// Mitsubishi GX Works2 project: BookEX6_29 Other   PLC: Q13UDV

// global labels: Global
VAR_GLOBAL
  bVar0 AT M5000 : BOOL;
  abArray0 AT M5010 : ARRAY [0..49] OF BOOL;
  sStr0 AT D5000 : STRING[199];
  sStr1 AT D5100 : STRING[199];
  sStr2 AT D5200 : STRING[199];
  sStr3 AT D5300 : STRING[199];
  sStr4 AT D5400 : STRING[199];
  sStr5 AT D5500 : STRING[199];
  sStr6 AT D5600 : STRING[199];
  sStr7 AT D5700 : STRING[199];
  sStr8 AT D5800 : STRING[199];
  sStr9 AT D5900 : STRING[199];
  iVar0 AT D4500 : INT;
  iVar1 AT D4501 : INT;
  iVar2 AT D4502 : INT;
  iVar3 AT D4503 : INT;
  iVar4 AT D4504 : INT;
  iVar5 AT D4505 : INT;
  iVar6 AT D4506 : INT;
  iVar7 AT D4507 : INT;
  iVar8 AT D4508 : INT;
  iVar9 AT D4509 : INT;
  dVar0 AT D4510 : DINT;
  dVar1 AT D4512 : DINT;
  dVar2 AT D4514 : DINT;
  dVar3 AT D4516 : DINT;
  dVar4 AT D4518 : DINT;
  dVar5 AT D4520 : DINT;
  dVar6 AT D4522 : DINT;
  dVar7 AT D4524 : DINT;
  dVar8 AT D4526 : DINT;
  dVar9 AT D4528 : DINT;
  wVar0 AT D4530 : WORD;
  wVar1 AT D4531 : WORD;
  wVar2 AT D4532 : WORD;
  wVar3 AT D4533 : WORD;
  wVar4 AT D4534 : WORD;
  wVar5 AT D4535 : WORD;
  wVar6 AT D4536 : WORD;
  wVar7 AT D4537 : WORD;
  wVar8 AT D4538 : WORD;
  wVar9 AT D4539 : WORD;
  dwVar0 AT D4540 : DWORD;
  dwVar1 AT D4542 : DWORD;
  dwVar2 AT D4544 : DWORD;
  dwVar3 AT D4546 : DWORD;
  dwVar4 AT D4548 : DWORD;
  dwVar5 AT D4550 : DWORD;
  dwVar6 AT D4552 : DWORD;
  dwVar7 AT D4554 : DWORD;
  dwVar8 AT D4556 : DWORD;
  dwVar9 AT D4558 : DWORD;
  fsVar0 AT D4560 : REAL;
  fsVar1 AT D4562 : REAL;
  fsVar2 AT D4564 : REAL;
  fsVar3 AT D4566 : REAL;
  fsVar4 AT D4568 : REAL;
  fsVar5 AT D4570 : REAL;
  fsVar6 AT D4572 : REAL;
  fsVar7 AT D4574 : REAL;
  fsVar8 AT D4576 : REAL;
  fsVar9 AT D4578 : REAL;
  fdVar0 AT D4580 : LREAL;
  tTime0 AT D4620 : TIME;
  tTime1 AT D4622 : TIME;
  tTime2 AT D4624 : TIME;
  tTime3 AT D4626 : TIME;
  tTime4 AT D4628 : TIME;
  tTime5 AT D4630 : TIME;
  tTime6 AT D4632 : TIME;
  tTime7 AT D4634 : TIME;
  tTime8 AT D4636 : TIME;
  tTime9 AT D4638 : TIME;
  tTime10 AT D4640 : TIME;
  bVar1 AT M5001 : BOOL;
  bVar2 AT M5002 : BOOL;
  bVar3 AT M5003 : BOOL;
  bVar4 AT M5004 : BOOL;
  bVar5 AT M5005 : BOOL;
  bVar6 AT M5006 : BOOL;
  bVar7 AT M5007 : BOOL;
  bVar8 AT M5008 : BOOL;
  bVar9 AT M5009 : BOOL;
  abArray1 AT M5060 : ARRAY [0..49] OF BOOL;
  abArray2 AT M5110 : ARRAY [0..49] OF BOOL;
  abArray3 AT M5160 : ARRAY [0..49] OF BOOL;
  abArray4 AT M5210 : ARRAY [0..49] OF BOOL;
  abArray5 AT M5260 : ARRAY [0..49] OF BOOL;
  abArray6 AT M5310 : ARRAY [0..49] OF BOOL;
  abArray7 AT M5360 : ARRAY [0..49] OF BOOL;
  abArray8 AT M5410 : ARRAY [0..49] OF BOOL;
  abArray9 AT M5460 : ARRAY [0..49] OF BOOL;
  fdVar1 AT D4584 : LREAL;
  fdVar2 AT D4588 : LREAL;
  fdVar3 AT D4592 : LREAL;
  fdVar4 AT D4596 : LREAL;
  fdVar5 AT D4600 : LREAL;
  fdVar6 AT D4604 : LREAL;
  fdVar7 AT D4608 : LREAL;
  fdVar8 AT D4612 : LREAL;
  fdVar9 AT D4616 : LREAL;
  afsPen0 AT D2000 : ARRAY [0..499] OF REAL;
  afsPen1 AT D3000 : ARRAY [0..499] OF REAL;
  abInp1 AT X10 : ARRAY [0..1] OF BOOL;
  abInp2 AT X12 : ARRAY [0..1] OF BOOL;
  adwD10 AT D10 : ARRAY [0..9] OF DWORD;
  awD10 AT D10 : ARRAY [0..19] OF WORD;
  abM10 AT M10 : ARRAY [0..19] OF BOOL;
END_VAR
// user libraries (not included): HMI

FUNCTION newENCO
VAR_INPUT
  w_IN : WORD;
END_VAR
VAR
  ix : INT;
  wTmp : WORD;
  iy : INT;
END_VAR
;
wTmp := H0001;
iy := 1;
FOR ix := 0 TO 15 DO 
	IF (w_IN AND wTmp) <> 0 THEN
		EXIT;
	END_IF;
	ROL(TRUE, 1, wTmp);
	iy := iy + 1;
END_FOR;
IF ix = 16 THEN
	iy := 0;
END_IF;
newENCO := iy;
END_FUNCTION

FUNCTION_BLOCK UpDw
VAR_INPUT
  b_CH1 : BOOL;
  b_CH2 : BOOL;
  b_RST : BOOL;
END_VAR
VAR_OUTPUT
  b_DIR : BOOL;
  i_Cnt : INT;
END_VAR
VAR
  bOld1 : BOOL;
  bOld2 : BOOL;
  bClk : BOOL;
  bClk1 : BOOL;
  baxb : BOOL;
  bClk2 : BOOL;
END_VAR
;
baxb := b_CH1 XOR b_CH2;
bClk1 := b_CH1 XOR bOld1;
bOld1 := b_CH1;
bClk2 := b_CH2 XOR bOld2;
bOld2 := b_CH2;
bClk := bClk1 OR bClk2;

IF baxb AND bClk1 THEN b_DIR := TRUE; END_IF;
IF baxb AND bClk2 THEN b_DIR := FALSE; END_IF;

IF bClk AND b_DIR THEN i_Cnt := i_Cnt + 1; END_IF;
IF bClk AND NOT b_DIR THEN i_Cnt := i_Cnt -1; END_IF;

IF b_RST THEN i_Cnt := 0; END_IF;
END_FUNCTION_BLOCK

PROGRAM Ex
(* structured ladder/FBD written out as ST: instructions are called as NAME(EN, inputs, outputs); _pN, _eN, _tN stand for wires *)
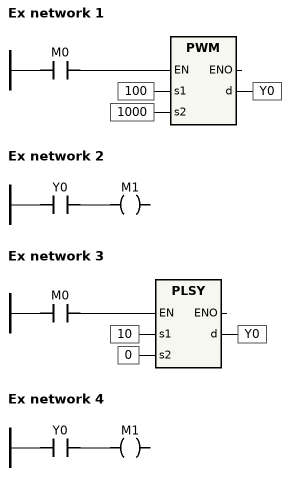
(* network 1 *)
PWM(M0, 100, 1000, Y0);
(* network 2 *)
M1 := Y0;
(* network 3 *)
PLSY(M0, 10, 0, Y0);
(* network 4 *)
M1 := Y0;
END_PROGRAM

PROGRAM ExMTR
(* structured ladder/FBD written out as ST: instructions are called as NAME(EN, inputs, outputs); _pN, _eN, _tN stand for wires *)
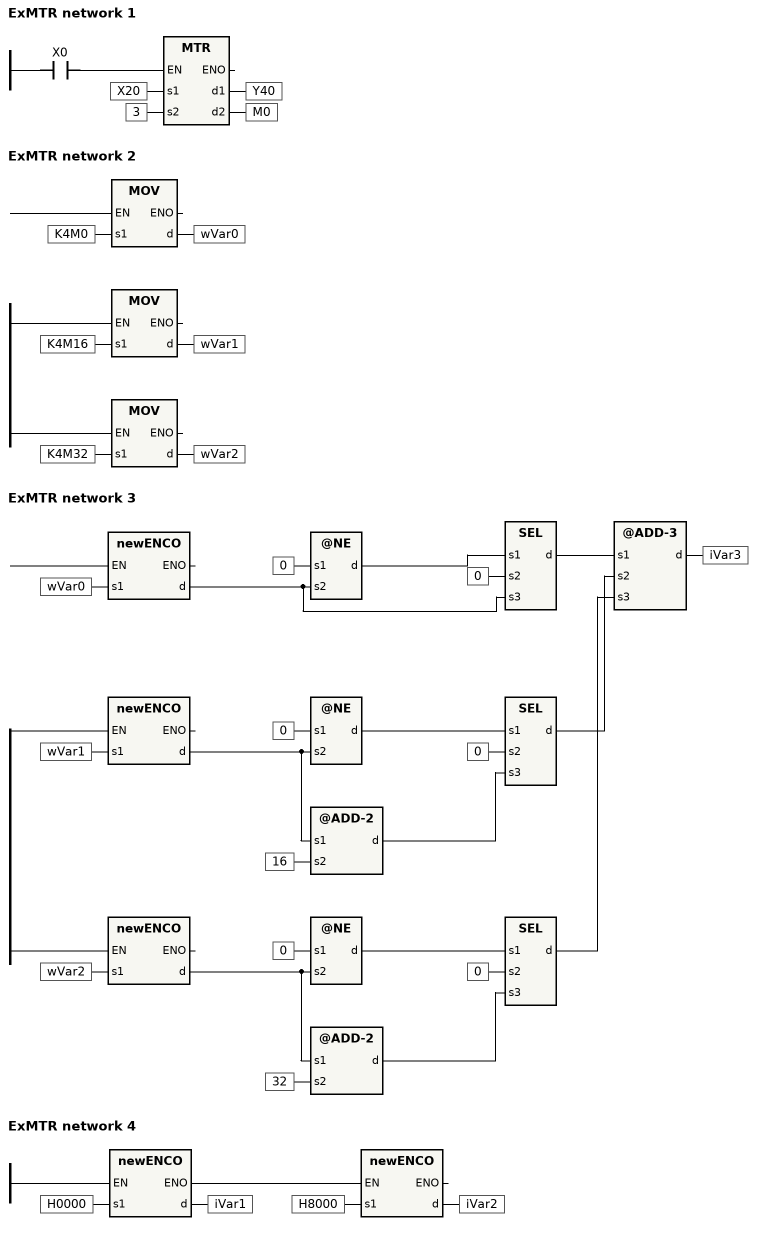
(* network 1 *)
MTR(X0, X20, 3, Y40, M0);
(* network 2 *)
MOV(TRUE, K4M0, wVar0);
MOV(TRUE, K4M16, wVar1);
MOV(TRUE, K4M32, wVar2);
(* network 3 *)
newENCO(TRUE, wVar0, _t1);
newENCO(TRUE, wVar1, _t2);
newENCO(TRUE, wVar2, _t3);
iVar3 := @ADD-3(SEL(@NE(0, _t1), 0, _t1), SEL(@NE(0, _t2), 0, @ADD-2(_t2, 16)), SEL(@NE(0, _t3), 0, @ADD-2(_t3, 32)));
(* network 4 *)
_e1 := newENCO(TRUE, H0000, iVar1);
newENCO(_e1, H8000, iVar2);
END_PROGRAM

PROGRAM ExPLSY
VAR
  HMI05_1 : HMI05;
END_VAR
(* structured ladder/FBD written out as ST: instructions are called as NAME(EN, inputs, outputs); _pN, _eN, _tN stand for wires *)
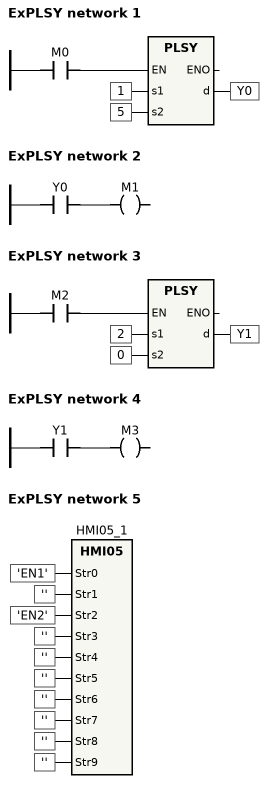
(* network 1 *)
PLSY(M0, 1, 5, Y0);
(* network 2 *)
M1 := Y0;
(* network 3 *)
PLSY(M2, 2, 0, Y1);
(* network 4 *)
M3 := Y1;
(* network 5 *)
HMI05_1(Str0 := 'EN1', Str1 := '', Str2 := 'EN2', Str3 := '', Str4 := '', Str5 := '', Str6 := '', Str7 := '', Str8 := '', Str9 := '');
END_PROGRAM

PROGRAM ExPWM
VAR
  HMI05_1 : HMI05;
  bFeed : BOOL;
  TON_HIGH_E_1 : TON_HIGH_E;
  TON_HIGH_E_2 : TON_HIGH_E;
END_VAR
(* structured ladder/FBD written out as ST: instructions are called as NAME(EN, inputs, outputs); _pN, _eN, _tN stand for wires *)
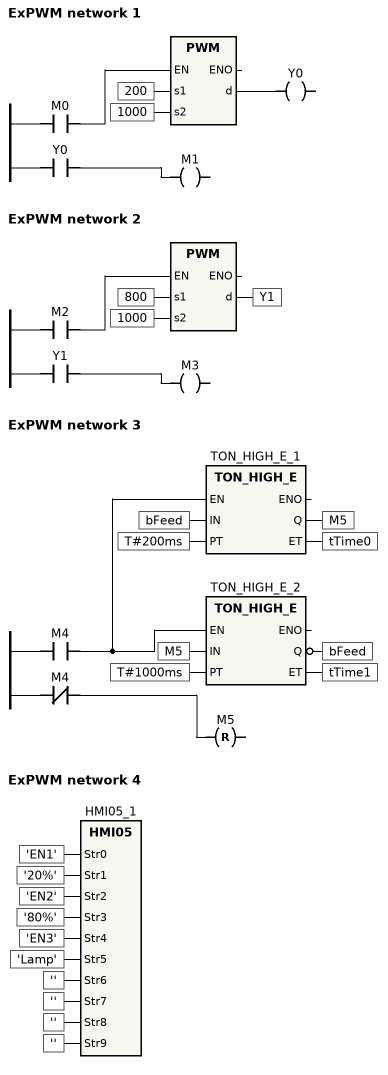
(* network 1 *)
PWM(M0, 200, 1000, _t1);
Y0 := _t1;
M1 := Y0;
(* network 2 *)
PWM(M2, 800, 1000, Y1);
M3 := Y1;
(* network 3 *)
TON_HIGH_E_1(EN := M4, IN := bFeed, PT := T#200ms, Q => M5, ET => tTime0);
TON_HIGH_E_2(EN := M4, IN := M5, PT := T#1000ms, ET => tTime1);
bFeed := NOT TON_HIGH_E_2.Q;
RST(NOT M4, M5);
(* network 4 *)
HMI05_1(Str0 := 'EN1', Str1 := '20%', Str2 := 'EN2', Str3 := '80%', Str4 := 'EN3', Str5 := 'Lamp', Str6 := '', Str7 := '', Str8 := '', Str9 := '');
END_PROGRAM

PROGRAM ExRAMP
VAR
  aiVar0 : ARRAY [0..1] OF INT;
  abRes3 : ARRAY [0..1] OF BOOL;
  HMI03_1 : HMI03;
END_VAR
(* structured ladder/FBD written out as ST: instructions are called as NAME(EN, inputs, outputs); _pN, _eN, _tN stand for wires *)
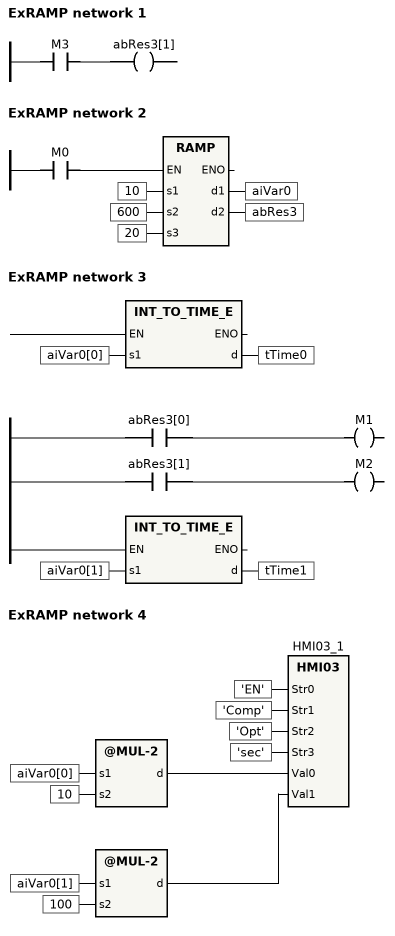
(* network 1 *)
abRes3[1] := M3;
(* network 2 *)
RAMP(M0, 10, 600, 20, aiVar0, abRes3);
(* network 3 *)
INT_TO_TIME_E(TRUE, aiVar0[0], tTime0);
INT_TO_TIME_E(TRUE, aiVar0[1], tTime1);
M1 := abRes3[0];
M2 := abRes3[1];
(* network 4 *)
HMI03_1(Str0 := 'EN', Str1 := 'Comp', Str2 := 'Opt', Str3 := 'sec', Val0 := @MUL-2(aiVar0[0], 10), Val1 := @MUL-2(aiVar0[1], 100));
END_PROGRAM

PROGRAM ExROTC
VAR
  aiVar2 : ARRAY [0..2] OF INT;
  abRes2 : ARRAY [0..7] OF BOOL;
  HMI05_1 : HMI05;
END_VAR
(* structured ladder/FBD written out as ST: instructions are called as NAME(EN, inputs, outputs); _pN, _eN, _tN stand for wires *)
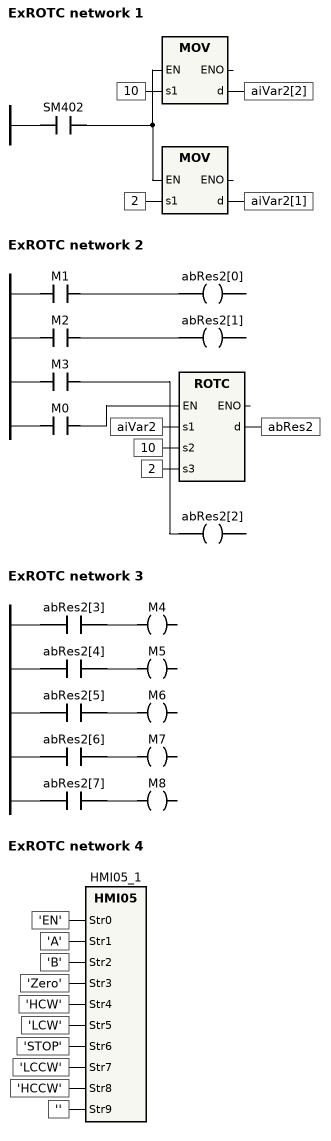
(* network 1 *)
MOV(SM402, 10, aiVar2[2]);
MOV(SM402, 2, aiVar2[1]);
(* network 2 *)
abRes2[0] := M1;
abRes2[1] := M2;
abRes2[2] := M3;
ROTC(M0, aiVar2, 10, 2, abRes2);
(* network 3 *)
M4 := abRes2[3];
M5 := abRes2[4];
M6 := abRes2[5];
M7 := abRes2[6];
M8 := abRes2[7];
(* network 4 *)
HMI05_1(Str0 := 'EN', Str1 := 'A', Str2 := 'B', Str3 := 'Zero', Str4 := 'HCW', Str5 := 'LCW', Str6 := 'STOP', Str7 := 'LCCW', Str8 := 'HCCW', Str9 := '');
END_PROGRAM

PROGRAM ExSPD
VAR
  HMI03_1 : HMI03;
END_VAR
(* structured ladder/FBD written out as ST: instructions are called as NAME(EN, inputs, outputs); _pN, _eN, _tN stand for wires *)
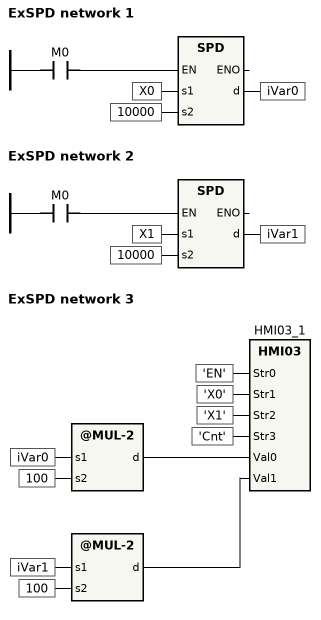
(* network 1 *)
SPD(M0, X0, 10000, iVar0);
(* network 2 *)
SPD(M0, X1, 10000, iVar1);
(* network 3 *)
HMI03_1(Str0 := 'EN', Str1 := 'X0', Str2 := 'X1', Str3 := 'Cnt', Val0 := @MUL-2(iVar0, 100), Val1 := @MUL-2(iVar1, 100));
END_PROGRAM

PROGRAM ExSTMR
VAR
  HMI05_1 : HMI05;
  abRes1 : ARRAY [0..3] OF BOOL;
END_VAR
(* structured ladder/FBD written out as ST: instructions are called as NAME(EN, inputs, outputs); _pN, _eN, _tN stand for wires *)
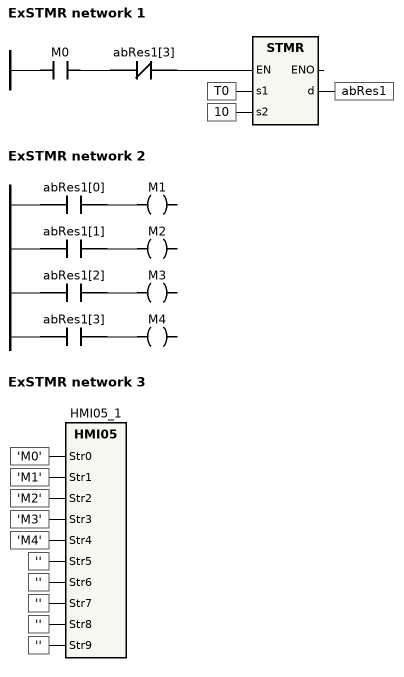
(* network 1 *)
STMR(M0 AND NOT abRes1[3], T0, 10, abRes1);
(* network 2 *)
M1 := abRes1[0];
M2 := abRes1[1];
M3 := abRes1[2];
M4 := abRes1[3];
(* network 3 *)
HMI05_1(Str0 := 'M0', Str1 := 'M1', Str2 := 'M2', Str3 := 'M3', Str4 := 'M4', Str5 := '', Str6 := '', Str7 := '', Str8 := '', Str9 := '');
END_PROGRAM

PROGRAM ExTTMR2
VAR
  aiVar0 : ARRAY [0..1] OF INT;
  HMI03_1 : HMI03;
  TTMR2_1 : TTMR2;
END_VAR
(* structured ladder/FBD written out as ST: instructions are called as NAME(EN, inputs, outputs); _pN, _eN, _tN stand for wires *)
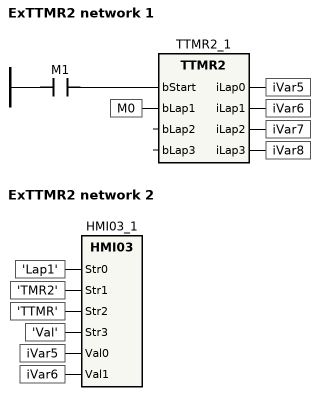
(* network 1 *)
TTMR2_1(bStart := M1, bLap1 := M0, iLap0 => iVar5, iLap1 => iVar6, iLap2 => iVar7, iLap3 => iVar8);
(* network 2 *)
HMI03_1(Str0 := 'Lap1', Str1 := 'TMR2', Str2 := 'TTMR', Str3 := 'Val', Val0 := iVar5, Val1 := iVar6);
END_PROGRAM

PROGRAM ExUDCNT
VAR
  HMI04_1 : HMI04;
END_VAR
(* structured ladder/FBD written out as ST: instructions are called as NAME(EN, inputs, outputs); _pN, _eN, _tN stand for wires *)
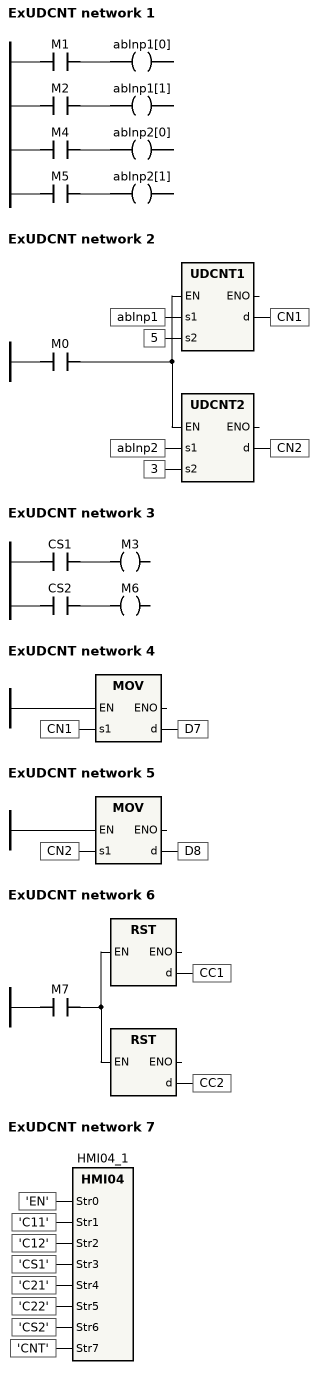
(* network 1 *)
abInp1[0] := M1;
abInp1[1] := M2;
abInp2[0] := M4;
abInp2[1] := M5;
(* network 2 *)
UDCNT1(M0, abInp1, 5, CN1);
UDCNT2(M0, abInp2, 3, CN2);
(* network 3 *)
M3 := CS1;
M6 := CS2;
(* network 4 *)
MOV(TRUE, CN1, D7);
(* network 5 *)
MOV(TRUE, CN2, D8);
(* network 6 *)
RST(M7, CC1);
RST(M7, CC2);
(* network 7 *)
HMI04_1(Str0 := 'EN', Str1 := 'C11', Str2 := 'C12', Str3 := 'CS1', Str4 := 'C21', Str5 := 'C22', Str6 := 'CS2', Str7 := 'CNT');
END_PROGRAM

PROGRAM ExUpDw
VAR
  HMI04_1 : HMI04;
  UpDw_1 : UpDw;
END_VAR
(* structured ladder/FBD written out as ST: instructions are called as NAME(EN, inputs, outputs); _pN, _eN, _tN stand for wires *)
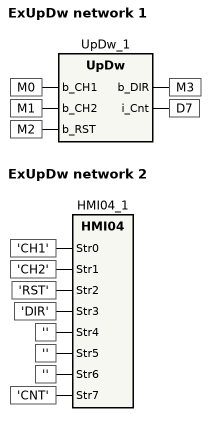
(* network 1 *)
UpDw_1(b_CH1 := M0, b_CH2 := M1, b_RST := M2, b_DIR => M3, i_Cnt => D7);
(* network 2 *)
HMI04_1(Str0 := 'CH1', Str1 := 'CH2', Str2 := 'RST', Str3 := 'DIR', Str4 := '', Str5 := '', Str6 := '', Str7 := 'CNT');
END_PROGRAM

PROGRAM ExTTMR
VAR
  aiVar0 : ARRAY [0..1] OF INT;
  HMI03_1 : HMI03;
  aiVar1 : ARRAY [0..1] OF INT;
END_VAR
(* structured ladder/FBD written out as ST: instructions are called as NAME(EN, inputs, outputs); _pN, _eN, _tN stand for wires *)
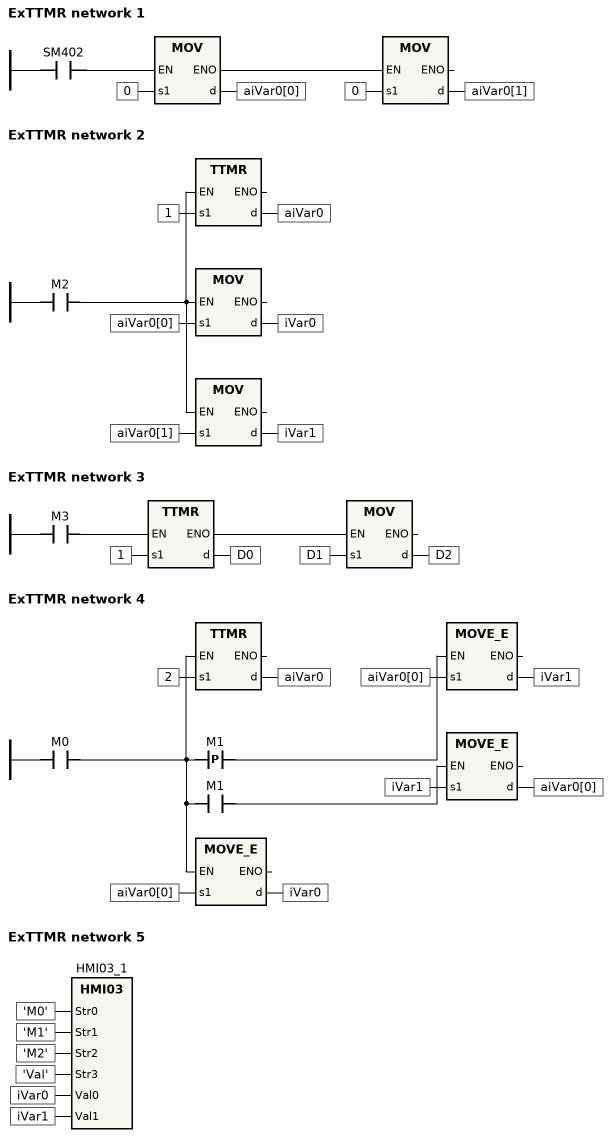
(* network 1 *)
_e1 := MOV(SM402, 0, aiVar0[0]);
MOV(_e1, 0, aiVar0[1]);
(* network 2 *)
TTMR(M2, 1, aiVar0);
MOV(M2, aiVar0[0], iVar0);
MOV(M2, aiVar0[1], iVar1);
(* network 3 *)
_e1 := TTMR(M3, 1, D0);
MOV(_e1, D1, D2);
(* network 4 *)
TTMR(M0, 2, aiVar0);
MOVE_E(M0, aiVar0[0], iVar0);
MOVE_E(M0 AND LDP(TRUE, M1), aiVar0[0], iVar1);
MOVE_E(M0 AND M1, iVar1, aiVar0[0]);
(* network 5 *)
HMI03_1(Str0 := 'M0', Str1 := 'M1', Str2 := 'M2', Str3 := 'Val', Val0 := iVar0, Val1 := iVar1);
END_PROGRAM

FUNCTION_BLOCK TTMR2
VAR_INPUT
  bStart : BOOL;
  bLap1 : BOOL;
  bLap2 : BOOL;
END_VAR
VAR_OUTPUT
  iLap0 : INT;
  iLap1 : INT;
  iLap2 : INT;
END_VAR
VAR
  dTime0 : DINT;
  dTime1 : DINT;
  dTime2 : DINT;
  dTmp : DINT;
END_VAR
VAR_OUTPUT
  iLap3 : INT;
END_VAR
VAR_INPUT
  bLap3 : BOOL;
END_VAR
VAR
  dTime3 : DINT;
END_VAR
;
IF LDP(TRUE, bStart) THEN
	dTime0 := 0;
	dTime1 := 0;
	dTime2 := 0;
	dTime3 := 0;
END_IF;
IF bStart THEN
	dTmp := INT_TO_DINT(SD520) *1000 + INT_TO_DINT(SD521);	
	dTime0 := dTime0 + dTmp;	
	IF LDP(TRUE, bLap1) THEN
		dTime1 := dTime0;
	END_IF;
	IF LDP(TRUE, bLap2) THEN
		dTime2 := dTime0;
	END_IF;
	IF LDP(TRUE, bLap3) THEN
		dTime3 := dTime0;
	END_IF;
END_IF;
iLap0 := DINT_TO_INT(dTime0 / 10000);	
iLap1 := DINT_TO_INT(dTime1 / 10000);
iLap2 := DINT_TO_INT(dTime2 / 10000);
iLap3 := DINT_TO_INT(dTime3 / 10000);
END_FUNCTION_BLOCK
